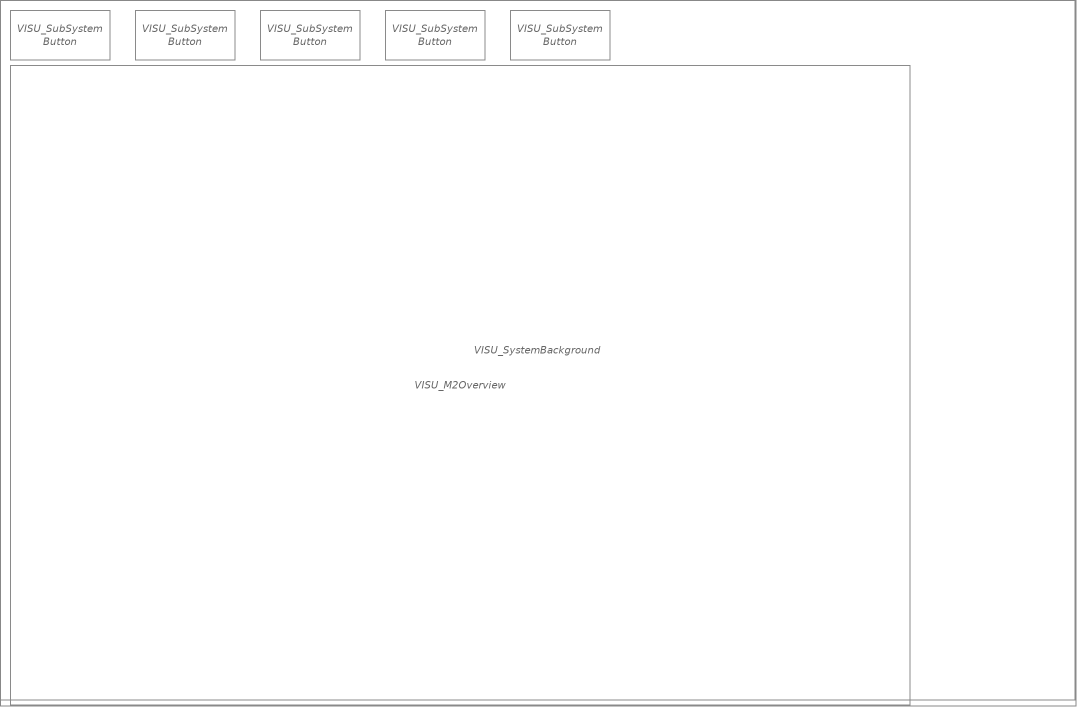
VISUALIZATION VISU_M2  // 1077x707
VAR_IN_OUT
	ref : M2;
	ref_io : M1M2IO;
    widget : M2Widget;
END_VAR
    Frame (0,0 1075x700)
        shows VISU_SystemBackground(color := widget.actualStatus.color)
    Frame (10,65 900x640)
        shows VISU_M2Overview(ref := ref, widget := widget)
        shows VISU_M2Axes(ref := ref, widget := widget)
        shows VISU_M2Technical(ref := ref, widget := widget)
        shows VISU_M1M2IO(ref := ref_io, widget := widget.io)
        shows VISU_M2Config(editableConfig := ref.editableConfig, activeConfig := ref.config, mgr := ref.parts.configManager, mgrWidget := widget.configManager, activeTab := widget.activeConfigTab, currentFocalStationPosition := widget.activeConfigFocalStation)
        p701045219: ref.editableConfig
        p2690442461: ref.config
        p942769723: ref.parts.configManager
        p2963374678: widget.configManager
        p459268616: widget
        p331394802: ref
        p3752816179: widget
        p2926564000: ref.editableConfig
        p430391093: ref.config
        p4084028830: ref.parts.configManager
        p721735225: widget.configManager
        p4165151898: widget.activeConfigTab
        p235284393: widget.activeConfigFocalStation
    Frame (10,10 100x50)
        shows VISU_SubSystemButton(widget := widget.button_overview)
        OnMouseClick: FrameSelectionChange Selection=SelectedFrame=b1e9e4b0-bf3d-440f-90c5-cb513105ccf1, GlobSel=AssignType=Directly, SelType=Locally
        OnMouseClick: execute { widget.activeTab := M2Tabs.OVERVIEW; }
    Frame (260,10 100x50)
        shows VISU_SubSystemButton(widget := widget.button_technical)
        OnMouseClick: FrameSelectionChange Selection=SelectedFrame=b1e9e4b0-bf3d-440f-90c5-cb513105ccf1, Selection=2, GlobSel=AssignType=Directly, SelType=Locally
        OnMouseClick: execute { widget.activeTab := M2Tabs.TECHNICAL; }
    Frame (385,10 100x50)
        shows VISU_SubSystemButton(widget := widget.button_io)
        OnMouseClick: FrameSelectionChange Selection=SelectedFrame=b1e9e4b0-bf3d-440f-90c5-cb513105ccf1, Selection=3, GlobSel=AssignType=Directly, SelType=Locally
        OnMouseClick: execute { widget.activeTab := M2Tabs.IO; }
    Frame (510,10 100x50)
        shows VISU_SubSystemButton(widget := widget.button_config)
        OnMouseClick: FrameSelectionChange Selection=SelectedFrame=b1e9e4b0-bf3d-440f-90c5-cb513105ccf1, Selection=4, GlobSel=AssignType=Directly, SelType=Locally
        OnMouseClick: execute { widget.activeTab := M2Tabs.CONFIG; }
    Frame (135,10 100x50)
        shows VISU_SubSystemButton(widget := widget.button_axes)
        OnMouseClick: FrameSelectionChange Selection=SelectedFrame=b1e9e4b0-bf3d-440f-90c5-cb513105ccf1, Selection=1, GlobSel=AssignType=Directly, SelType=Locally
        OnMouseClick: execute { widget.activeTab := M2Tabs.AXES; }
END_VISUALIZATION

(* stored: Version 1.1.0.1, ProductVersion 3.1.4019.2
   Visu VISU_M2: Id {c03627fa-5fd0-4cef-ac98-acfe91d7e836} *)
